DATA_BLOCK "ST10_StopperCtrl_DB"
VAR
  Stopper : Array[1..100] of "StopperCtrl";
END_VAR
BEGIN
END_DATA_BLOCK
